# EPICS autosave request: tomoScanApp/Db/tomoScan_prisma_settings.req
# This file is used by autosave to determine what PVs to save
# It is also used by tomoScan to determine what PVs to create

# This is the file for the tomoscan_prisma derived class.

#################
# Interlaced scan
#################
$(P)$(R)InterlacedScan
$(P)$(R)InterlacedFileName
$(P)$(R)StabilizationTime

#########################
# Beam status information
#########################
$(P)$(R)Testing
$(P)$(R)OpenShutter
$(P)$(R)CloseShutter

$(P)$(R)RotationEnd
